FUNCTION_BLOCK FB3_Modules
VAR_INPUT
END_VAR
VAR_OUTPUT
END_VAR
VAR
	newboxdump : MOD_InputBelt_Q_stRequest;
	WeighbridgeDefinitions : MOD_WeighBridge_I_stDefinitions;
END_VAR

Parts.Belt(iq_Commandstate := Parts.GlobalCommandState,
	q_NewBox => newboxdump);
	
WeighbridgeDefinitions.DetractorWeight := 60;
WeighbridgeDefinitions.OperatingWeight := 1000;
WeighbridgeDefinitions.WeightLimit := 6000; // needs to be set by external source like HMI	
Parts.Weighbridge(i_Definitions := WeighbridgeDefinitions,
	iq_CommandState  := Parts.GlobalCommandState);

Parts.Crane.i_Input.Ready := Parts.Belt.q_BoxReady.BoxReady;
Parts.Crane(i_LoadGrabbed := Parts.MechanicalGrabCrane.q_Grabbed,
	q_Grab => Parts.MechanicalGrabCrane.i_Grab,
	iq_CommandState  := Parts.GlobalCommandState);
	
Parts.MechanicalGrabCrane(iq_CommandState  := Parts.GlobalCommandState);

END_FUNCTION_BLOCK

(* stored: Version 1.1.0.1, ProductVersion 3.1.4024.6
   POU FB3_Modules: Id {54cc7670-8201-4bdf-a347-fc97717409df}, SpecialFunc None *)
